FUNCTION_BLOCK FbStartStopCircuit
VAR_INPUT
	xStart: BOOL;
	xStop: BOOL;
END_VAR
VAR_OUTPUT
	xRun: BOOL;
END_VAR

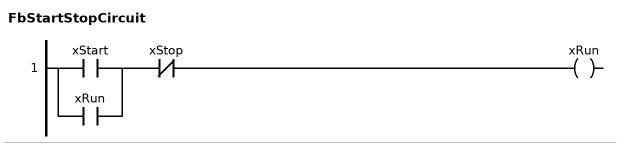
// NETWORK 1
xRun := (xStart OR xRun) AND NOT xStop;

END_FUNCTION_BLOCK

(* stored: Version 1.1.0.1, ProductVersion 3.1.4024.12
   POU FbStartStopCircuit: Id {df4faf84-33a2-44f0-88db-c04736871021}, SpecialFunc None *)
